PROGRAM MAIN
VAR
	s_ParamPathnames	: ARRAY[1..Param_Project.n_MaxParamFolders] OF STRING := ['C:\Cleanroom_Connect\Parameters'];//, 'C:\Cleanroom_Connect\Param\DockingInterface'];

	User : STRING := '<user_name>';
	SoftwareVersion : STRING := '<software_version>';
	InitDone : BOOL;
	Shutdown : BOOL;
	
//--	fbHmiParamHandler : FB_HmiParamHandler;
//--	fbHmiParamHandler_1 : FB_HmiParamHandler;
//--	fbHmiParamHandler_2 : FB_HmiParamHandler;
//--	fbHmiParamHandler_3 : FB_HmiParamHandler;
	
//--	arr_sValue : ARRAY[1..3] OF STRING;
//--	arr_fValue : ARRAY[1..3] OF LREAL;
	
//--ncTest : NC_Test;	

	//..
//--	fbMovAvg : FB_MovAvg;
	
//--	fbHAL : HAL;
	
//--	{attribute 'TcLinkTo' := 'TIID^Master (EtherCAT)^Term 1 (EK1200)^Term 9 (EL1809)^Channel 1^Input'}
//--	//--bVarIn2    AT%I*  : BOOL;  // linked via attribute
//--	GVL_Modules_g_emDockingInterface_s_cmDockingClampsUpper_I_bStaValveIsOn    AT%I*  : BOOL;  // linked via attribute 

//--	{attribute 'TcLinkTo' := 'TIID^Master (EtherCAT)^Term 1 (EK1200)^Term 9 (EL1809)^Channel 2^Input'}
//--	GVL_Modules_g_emUtilities_s_diSafetyOk_I_bStaInput AT%I* : BOOL;
	
//--	{attribute 'TcLinkTo' := 'TIID^Master (EtherCAT)^Term 1 (EK1200)^Term 9 (EL1809)^Channel 3^Input'}
//--	GVL_Modules_g_emUtilities_s_diPowerOk_I_bStaInput AT%I* : BOOL;
	
//--	{attribute 'TcLinkTo' := 'TIID^Master (EtherCAT)^Term 1 (EK1200)^Term 9 (EL1809)^Channel 4^Input'}
//--	GVL_Modules_g_emUtilities_s_diAirPressureOk_I_bStaInput AT%I* : BOOL;
	
END_VAR


//--ncTest();

GVL_KMWEGenericLib.g_fbAlarmManager();


GVL_KMWEGenericLib.g_fbParamManager.p_bShowHmiParam := TRUE;

GVL_KMWEGenericLib.g_fbParamManager(
	i_sPathName := s_ParamPathnames, 
	i_osrResetImportExport := GVL_KMWEGenericLib.g_fbAlarmManager.p_osrReset);
	
GVL.g_unCleanroomConnect.p_bCmdReset := GVL_KMWEGenericLib.g_fbAlarmManager.p_osrReset;
GVL.g_unCleanroomConnect();

//--//Just a test
//--fbMovAvg(
//--	i_rIn := ,
//--	i_nSamples := , 
//--	o_rOut=> );

//--fbHAL();

//Test parameter handling
(*
fbHmiParamHandler(
	i_fDefaultValue := ,
	i_sName := 'Name',
	i_nArrayFolderIndex := 1,
	i_bIsNumber := FALSE);

fbHmiParamHandler_1(
	i_fDefaultValue := ,
	i_sName := 'Param 1',
	i_nArrayFolderIndex := 1,
	i_bIsNumber := TRUE);
	
fbHmiParamHandler_2(
	i_fDefaultValue := ,
	i_sName := 'Param 2',
	i_nArrayFolderIndex := 1,
	i_bIsNumber := TRUE);
	
fbHmiParamHandler_3(
	i_fDefaultValue := ,
	i_sName := 'Param 3',
	i_nArrayFolderIndex := 1,
	i_bIsNumber := TRUE);
	
arr_sValue[1] := fbHmiParamHandler.p_sValue;
arr_fValue[1] := fbHmiParamHandler_1.p_fValue;
arr_fValue[2] := fbHmiParamHandler_2.p_fValue;
arr_fValue[3] := fbHmiParamHandler_3.p_fValue;
	
*)

END_PROGRAM

(* stored: Version 1.1.0.1, ProductVersion 3.1.4024.12
   POU MAIN: Id {c137dca6-2078-4081-8260-8d6099001278}, SpecialFunc None *)
